TYPE ST_CartMotorOutput  :
STRUCT
	//MingZhi drive ues
	m_cmdVelMz:DINT:=0;
	
	m_cmdAccMz:DINT:=0;
	
	m_cmdVelMzVelMode:DINT:=0;
	
	
END_STRUCT
END_TYPE

(* stored: Version 1.1.0.1, ProductVersion 3.1.4024.11
   DUT ST_CartMotorOutput: Id {469bcf24-d774-4d2a-9283-c2c92d1096c7} *)
